// Mitsubishi GX Works2 project: IHW3   PLC: Q03UDE

// global labels: Global1
VAR_GLOBAL
  STARTBUTTON AT X40 : BOOL;
  STOPBUTTON AT X41 : BOOL;
  ESTOPBUTTON AT X42 : BOOL;
  DTRUONG AT Y50 : BOOL;
  DDAI AT Y51 : BOOL;
  DHOC AT Y52 : BOOL;
  DCONG AT Y53 : BOOL;
  DNGHIEP AT Y54 : BOOL;
  DHA AT Y55 : BOOL;
  DNOI AT Y56 : BOOL;
END_VAR

PROGRAM MAIN
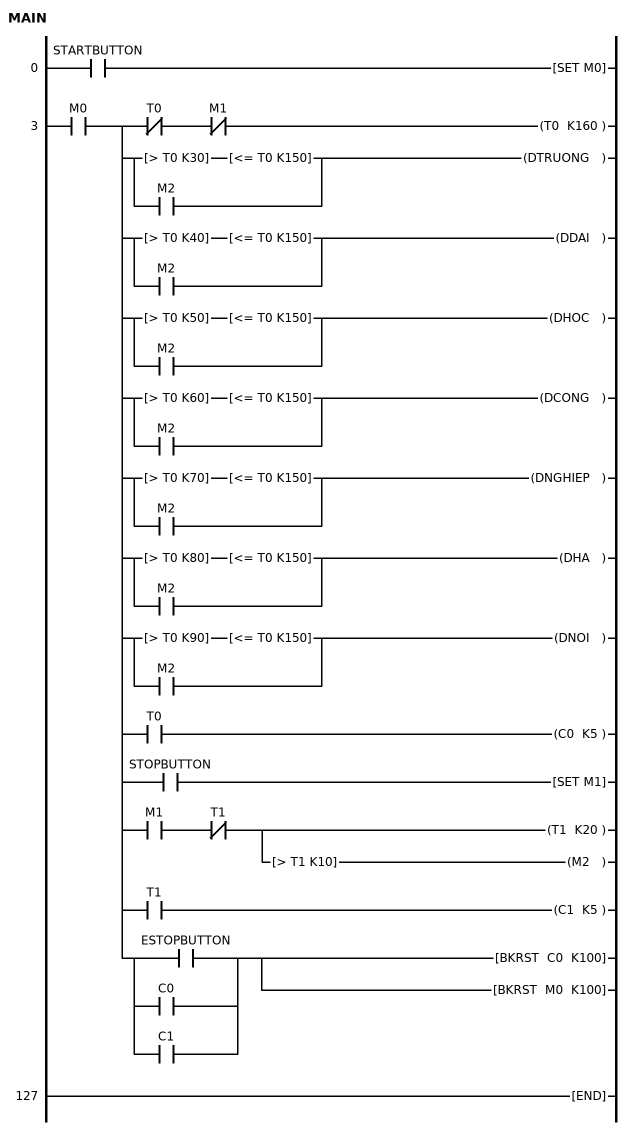
0     LD      STARTBUTTON
      SET     M0
3     LD      M0
      MPS
      ANI     T0
      ANI     M1
      OUT     T0 K160
      MRD
      LD>     T0 K30
      AND<=   T0 K150
      OR      M2
      ANB
      OUT     DTRUONG
      MRD
      LD>     T0 K40
      AND<=   T0 K150
      OR      M2
      ANB
      OUT     DDAI
      MRD
      LD>     T0 K50
      AND<=   T0 K150
      OR      M2
      ANB
      OUT     DHOC
      MRD
      LD>     T0 K60
      AND<=   T0 K150
      OR      M2
      ANB
      OUT     DCONG
      MRD
      LD>     T0 K70
      AND<=   T0 K150
      OR      M2
      ANB
      OUT     DNGHIEP
      MRD
      LD>     T0 K80
      AND<=   T0 K150
      OR      M2
      ANB
      OUT     DHA
      MRD
      LD>     T0 K90
      AND<=   T0 K150
      OR      M2
      ANB
      OUT     DNOI
      MRD
      AND     T0
      OUT     C0 K5
      MRD
      AND     STOPBUTTON
      SET     M1
      MRD
      AND     M1
      ANI     T1
      OUT     T1 K20
      AND>    T1 K10
      OUT     M2
      MRD
      AND     T1
      OUT     C1 K5
      MPP
      LD      ESTOPBUTTON
      OR      C0
      OR      C1
      ANB
      BKRST   C0 K100
      BKRST   M0 K100
127   END
END_PROGRAM
